// SIMATIC S7-200 project (STEP 7-Micro/WIN), CPU 226 REL 02.00

ORGANIZATION_BLOCK MAIN:OB1
TITLE=【PLC程序案例教程免烧砖机】
// 此PLC程序控制免烧砖机，包含生产控制和故障处理模块。 系统通过原料输送带、模具和成品输送带运行。
// 系统部署在生产车间，通过触摸屏操作界面进行参数设置和状态监控，支持手动和自动两种模式，满足不同操作需求。
// 
// 
// 操作员按下点动按钮可启动成品输送带。系统通过模式标志切换手动和自动模式：当模式标志为0时，系统处于手动模式；当模式标志为1时，系统处于自动模式。
// 在自动模式下，操作员按下启动按钮启动生产流程。系统首先检查生产批次计数器是否大于0，并确保到位传感器1、到位传感器3、到位传感器4和到位传感器5全部检测到位，只有这些条件满足时，状态变量才会从100变为58，进入生产状态。若任一传感器未就位，系统保持待机，避免设备运行风险。
// 生产开始后，原料通过输送带输入，随后进入布料阶段。布料过程被调用，当布料传感器检测到原料到位时，置位布料标志。在布料过程中，若布料标志置位，则激活布料执行信号。布料过程中，布料计数器记录布料次数。系统将布料计数器与布料上限计数器比较。若布料计数器小于布料上限计数器，布料继续；若达到上限，则根据布料模式变量切换布料逻辑，确保原料分配精准。
// 布料完成后，系统进入压制阶段，置位压制控制标志和压制执行信号。压制动作持续进行，直到到位传感器2检测到模具到位，随后压制执行信号复位。压制开始后，压制定时器1控制初始压制时间。随后，压制定时器2进一步控制压制时间，确保砖块成型质量稳定。压制结束后，成品通过成品输送带输出。压制计数器记录压制次数。系统将压制计数器与目标压制计数器比较以跟踪生产进度。
// 在手动模式下，操作员可通过点动按钮启动成品输送带。当到位传感器5置位时，成品输送带停止运行，以防止误操作导致设备损坏或安全事故。
// 系统还具备完善的故障监控功能。若故障总标志置位，表明某个环节出现异常，故障显示位1或故障显示位2会具体指示故障源，如执行机构1或2的异常状态。操作员可通过触摸屏查看详细故障信息并采取措施。
// 
BEGIN
Network 1 // 网络标题
// 网络注释
LD     SM0.1
CALL   SYSRESET:SBR13
Network 2
LDN    M31.0
CALL   Trouble_Display:SBR1
CALL   Run_Data_Change:SBR6
Network 3
LDN    M31.0
CALL   Trou_Run:SBR18
Network 4
LD     SM0.0
CALL   IOContral:SBR3
CALL   TOUCHER:SBR12
CALL   TOUCHER_Time:SBR10
CALL   TOUCHER_Time1:SBR11
CALL   SETUP_DATE:SBR19
Network 5
LDN    M3.2
AN     M31.0
CALL   Manual_batch:SBR4
CALL   Spot_Batch:SBR0
Network 6
LDN    M3.2
AN     M31.0
CALL   Manual_Spot:SBR17
Network 7
LD     M3.2
A      I2.3
AN     M31.0
CALL   AUTO_RESET:SBR5
CALL   Send_Take:SBR22
CALL   AUTO_PRODUCT:SBR15
Network 8
LDN    I4.0
CALL   Manual_batch1:SBR7
Network 9
LD     I4.0
CALL   AUTO1:SBR8
END_ORGANIZATION_BLOCK

SUBROUTINE_BLOCK Spot_Batch:SBR0
TITLE=子程序注释
BEGIN
Network 1 // 网络标题
// 网络注释
LDN    M4.4
AB=    VB742, 10
LD     I0.7
O      M22.5
ALD
AN     M8.0
S      M4.4, 1
S      M10.1, 1
Network 2
LD     M4.4
LDN    M22.5
AN     I0.7
O      M8.0
OB=    VB742, 0
ALD
R      M10.1, 1
R      M4.4, 1
Network 3
LDN    M4.7
AB=    VB742, 10
LD     I1.0
O      M22.6
ALD
AN     I3.2
S      M4.7, 1
S      M10.0, 1
Network 4
LD     M4.7
LDN    M22.6
AN     I1.0
O      I3.2
OB=    VB742, 0
ALD
R      M10.0, 1
R      M4.7, 1
Network 5
LDN    M5.1
LD     I0.5
O      M22.3
ALD
AB=    VB742, 10
AN     I2.4
AN     M8.2
S      M5.1, 1
S      M10.2, 1
Network 6
LD     M5.1
LDN    M22.3
AN     I0.5
O      M8.2
O      I2.4
OB=    VB742, 0
ALD
R      M10.2, 1
R      M5.1, 1
Network 7
LDN    M5.3
AB=    VB742, 10
LD     I0.6
O      M22.4
ALD
AN     I2.5
S      M5.3, 1
S      M10.4, 1
Network 8
LD     M5.3
LDN    M22.4
AN     I0.6
O      I2.5
OB=    VB742, 0
ALD
R      M10.4, 1
R      M5.3, 1
Network 9
LDN    M6.5
AB=    VB742, 10
LD     I1.1
O      M22.7
ALD
AN     I2.6
AN     M9.0
S      M6.5, 1
S      M11.4, 1
Network 10
LD     M6.5
LDN    M22.7
AN     I1.1
O      M9.0
O      I2.6
OB=    VB742, 0
ALD
R      M11.4, 1
R      M6.5, 1
Network 11
LDN    M6.7
AB=    VB742, 10
LD     I1.2
O      M23.0
ALD
AN     I2.7
AN     M9.1
S      M6.7, 1
S      M11.6, 1
Network 12
LD     M6.7
LDN    M23.0
AN     I1.2
O      M9.1
O      I2.7
OB=    VB742, 0
ALD
R      M11.6, 1
R      M6.7, 1
Network 13
LDN    M7.1
AB=    VB742, 10
LD     I1.3
O      M23.1
ALD
AN     I3.0
AN     M9.2
S      M7.1, 1
S      M12.1, 1
Network 14
LD     M7.1
LDN    M23.1
AN     I1.3
O      M9.2
O      I3.0
OB=    VB742, 0
ALD
R      M12.1, 1
R      M7.1, 1
Network 15
LDN    M7.3
AB=    VB742, 10
LD     I1.4
O      M23.2
ALD
AN     I3.1
AN     M9.3
S      M7.3, 1
S      M12.3, 1
Network 16
LD     M7.3
LDN    M23.2
AN     I1.4
O      M9.3
O      I3.1
OB=    VB742, 0
ALD
R      M12.3, 1
R      M7.3, 1
Network 17
LDN    M7.5
AB=    VB742, 10
LD     I1.5
O      M23.3
ALD
AN     I2.7
AN     M12.6
S      M7.5, 1
S      M12.0, 1
Network 18
LD     M7.5
LDN    M23.3
AN     I1.5
O      M12.6
O      I2.7
OB=    VB742, 0
ALD
R      M12.0, 1
R      M7.5, 1
END_SUBROUTINE_BLOCK

SUBROUTINE_BLOCK Trouble_Display:SBR1
TITLE=
BEGIN
Network 1
LD     I0.7
O      M22.5
AN     I2.5
AN     V5000.3
AB=    VB742, 0
=      V5000.3
Network 2
LD     I1.0
O      M22.6
A      I3.2
AN     V5000.4
=      V5000.4
Network 3
LD     I0.5
O      M22.3
LD     I2.4
ON     I3.2
ON     I2.6
ON     I3.1
ALD
AN     V5000.5
AB=    VB742, 0
=      V5000.5
Network 4
LD     I0.6
O      M22.4
LDN    I2.6
O      I2.5
ALD
AN     V5000.6
AB=    VB742, 0
=      V5000.6
Network 5
LD     I1.1
O      M22.7
A      I2.6
AN     V5001.3
=      V5001.3
Network 6
LD     I1.2
O      M23.0
LDN    I2.5
O      I2.7
ALD
AN     V5001.4
AB=    VB742, 0
=      V5001.4
Network 7
LD     I1.5
O      M23.3
LDN    I2.5
O      I2.7
ALD
AN     V5001.5
AB=    VB742, 0
=      V5001.5
Network 8
LD     I1.4
O      M23.2
A      I3.1
AN     V5001.6
=      V5001.6
Network 9
LD     I1.3
O      M23.1
LDN    I2.5
O      I3.0
ALD
AN     V5001.7
AB=    VB742, 0
=      V5001.7
Network 10
LD     I0.5
O      M22.3
LD     I0.6
O      M22.4
ALD
=      V5003.3
Network 11
LD     I1.1
O      M22.7
LD     I1.2
O      M23.0
ALD
=      V5003.4
Network 12
LD     I1.3
O      M23.1
LD     I1.4
O      M23.2
ALD
=      V5003.5
END_SUBROUTINE_BLOCK

SUBROUTINE_BLOCK RESET:SBR2
TITLE=
BEGIN
Network 1
LD     SM0.0
R      M3.3, 1
Network 2
LD     SM0.0
MOVB   100, VB700
MOVB   100, VB702
Network 3
LD     SM0.0
MOVB   0, QB0
MOVB   0, QB2
Network 4
LD     SM0.0
R      Q1.3, 1
R      Q1.4, 1
R      Q1.5, 1
R      Q1.6, 1
R      Q1.7, 1
Network 5
LD     SM0.0
MOVW   +0, VW802
MOVW   +0, VW806
MOVW   +0, VW812
Network 6
LD     SM0.0
R      M10.0, 6
R      M11.4, 4
R      M12.0, 8
R      M30.0, 1
R      M18.1, 1
R      M18.4, 1
R      M28.7, 1
Network 7
LD     SM0.0
R      M18.7, 1
R      V5003.7, 3
R      M21.0, 4
R      V5003.1, 2
R      M2.3, 1
Network 8
LD     SM0.0
R      M2.0, 3
R      M4.4, 1
R      M4.7, 1
R      M5.1, 1
R      M5.3, 1
R      M6.5, 1
R      M6.7, 1
R      M7.1, 1
R      M7.3, 1
R      M7.5, 1
R      M18.0, 2
R      M18.5, 1
Network 9
LD     SM0.0
R      M4.2, 1
R      M4.5, 1
R      M5.0, 1
R      M5.2, 1
R      M6.4, 1
R      M6.6, 1
R      M7.0, 1
R      M7.2, 1
R      M7.6, 1
R      M12.7, 1
R      M7.4, 1
R      M7.7, 1
R      M18.2, 3
R      M4.3, 1
R      M4.6, 1
Network 10
LD     SM0.0
R      M21.6, 1
R      M29.0, 8
R      M30.3, 5
END_SUBROUTINE_BLOCK

SUBROUTINE_BLOCK IOContral:SBR3
TITLE=
BEGIN
Network 1
LD     SM0.0
TODR   VB5100
BMB    VB5100, VB2450, 8
Network 2
LD     SM0.0
LPS
A      M31.1
AW<=   VW94, VW82
R      M31.0, 1
LRD
A      M31.1
AW>    VW94, VW82
S      M31.0, 1
LRD
A      M31.2
AW<=   VW94, VW86
R      M31.0, 1
LRD
A      M31.2
AW>    VW94, VW86
S      M31.0, 1
LPP
AW=    VW90, +370
R      M31.0, 1
Network 3
LDW>=  VW804, +1
MOVW   VW804, VW800
-I     +1, VW800
Network 4
LDB=   QB0, 0
MOVW   +0, VW144
MOVW   +0, VW146
Network 5
LD     I2.3
A      Q1.2
MOVW   VW144, VW136
*I     VW152, VW136
MOVW   VW146, VW138
*I     VW148, VW138
Network 6
LD     M4.0
LD     I0.4
O      M22.2
ALD
ED
R      M4.0, 2
R      Q1.2, 1
Network 7
LD     M4.0
A      M4.1
AN     I2.3
R      M4.0, 2
R      Q1.2, 1
S      M3.0, 1
R      M3.1, 1
CALL   RESET:SBR2
Network 8
LD     Q1.2
A      I2.3
AN     M4.1
S      M4.1, 1
Network 9
LDN    M4.0
AN     I2.3
LD     I0.4
O      M22.2
ALD
ED
S      M4.0, 1
S      Q1.2, 1
Network 10
LD     I2.3
A      Q1.2
MOVW   VW136, AQW0
MOVW   VW138, AQW2
Network 11
LD     M31.0
LD     I0.3
O      I0.5
O      I0.6
O      I0.7
O      I1.0
O      I1.1
O      I1.2
O      I1.3
O      I1.4
O      I1.5
O      I1.6
O      I1.7
O      I2.0
O      I2.1
ALD
=      V5005.4
Network 12
LDN    M31.0
A      I0.0
AN     I2.3
LD     I0.3
O      I0.5
O      I0.6
O      I0.7
O      I1.0
O      I1.1
O      I1.2
O      I1.3
O      I1.4
O      I1.5
ALD
=      V5005.3
Network 13
LDN    M31.0
AN     M3.1
AN     V5003.6
LD     I0.3
O      M22.1
ALD
LD     M3.3
ON     M3.2
ON     I2.5
ON     I2.3
ON     I3.3
ON     I2.6
ON     I3.1
ALD
=      V5003.6
Network 14
LDW<>  VW90, +370
AN     M28.5
A      M28.6
LPS
INCW   VW1006
AENO
MOVW   VW1006, VW94
LRD
S      M28.5, 1
LPP
R      M28.6, 1
Network 15
LD     M28.5
AN     SM31.7
R      SM31.0, 1
S      SM31.1, 1
MOVW   +94, SMW32
S      SM31.7, 1
R      M28.5, 1
Network 16
LD     M3.6
R      M3.1, 1
S      M3.0, 1
R      M3.6, 1
CALL   RESET:SBR2
Network 17
LD     M3.5
R      M3.5, 1
CALL   RESET:SBR2
Network 18
LD     M3.1
LD     M9.3
O      M8.1
O      M8.2
O      M8.3
O      M9.0
O      M9.2
O      M12.6
O      M9.7
O      M9.1
ALD
S      M3.0, 1
R      M3.1, 1
CALL   RESET:SBR2
Network 19
LD     M3.7
AN     I4.0
CALL   RESET1:SBR9
Network 20
LDN    I0.0
S      M3.4, 1
Network 21
LD     I0.0
LPS
R      M3.4, 1
EU
S      M3.5, 1
LPP
ED
S      M3.6, 1
Network 22
LDN    M3.4
S      M3.2, 1
Network 23
LD     M3.4
R      M3.2, 1
Network 24
LDN    I4.0
R      M3.7, 1
Network 25
LD     I4.0
S      M3.7, 1
END_SUBROUTINE_BLOCK

SUBROUTINE_BLOCK Manual_batch:SBR4
TITLE=
BEGIN
Network 1
LD     I0.2
O      M22.0
CALL   RESET:SBR2
Network 2
LD     M4.2
AB=    VB742, 0
A      Q0.3
LD     I0.7
O      M22.5
ALD
ED
R      M10.1, 1
R      M4.2, 1
Network 3
LD     M4.2
A      Q0.3
LD     M8.0
ON     I2.5
O      I1.0
OB=    VB742, 10
O      M22.6
ALD
R      M10.1, 1
R      M4.2, 1
Network 4
LDN    M4.2
AN     M4.3
A      I2.5
AB=    VB742, 0
AN     M8.0
AN     M22.6
AN     I1.0
LD     I0.7
O      M22.5
ALD
ED
S      M4.2, 1
S      M10.1, 1
R      T163, 1
Network 5
LD     M4.5
AB=    VB742, 0
A      Q0.2
LD     I1.0
O      M22.6
ALD
ED
R      M10.0, 1
R      M4.5, 1
Network 6
LD     M4.5
A      Q0.2
LD     I3.2
O      M8.1
O      I0.7
OB=    VB742, 10
O      M22.5
ALD
R      M10.0, 1
R      M4.5, 1
Network 7
LDN    M4.5
AN     M4.3
AN     M22.5
AN     I0.7
AB=    VB742, 0
AN     M8.1
AN     I3.2
LD     I1.0
O      M22.6
ALD
ED
S      M4.5, 1
S      M10.0, 1
Network 8
LD     M5.0
AB=    VB742, 0
A      Q0.1
LD     I0.5
O      M22.3
ALD
ED
R      M10.2, 1
R      M5.0, 1
Network 9
LD     M5.0
A      Q0.1
LD     I2.4
O      M8.2
O      M22.4
ON     I3.2
ON     I2.6
ON     I3.1
O      I0.6
OB=    VB742, 10
ALD
R      M10.2, 1
R      M5.0, 1
Network 10
LDN    M5.0
AB=    VB742, 0
A      I3.2
A      I2.6
A      I3.1
AN     M22.4
AN     I0.6
AN     I2.4
AN     M8.2
LD     I0.5
O      M22.3
ALD
ED
S      M5.0, 1
S      M10.2, 1
Network 11
LD     M5.2
AB=    VB742, 0
A      Q0.0
LD     I0.6
O      M22.4
ALD
ED
R      M10.4, 1
R      M5.2, 1
Network 12
LD     M5.2
A      Q0.0
LD     I2.5
O      M8.3
ON     I2.6
O      I0.5
OB=    VB742, 10
O      M22.3
ALD
R      M10.4, 1
R      M5.2, 1
Network 13
LDN    M5.2
AB=    VB742, 0
A      I2.6
AN     I2.5
AN     M22.3
AN     I0.5
AN     M8.3
LD     I0.6
O      M22.4
ALD
ED
S      M5.2, 1
S      M10.4, 1
Network 14
LD     M6.4
AB=    VB742, 0
A      Q0.4
LD     I1.1
O      M22.7
ALD
ED
R      M11.4, 1
R      M6.4, 1
Network 15
LD     M6.4
A      Q0.4
LD     I2.6
O      M9.0
O      I1.2
OB=    VB742, 10
O      M23.0
ALD
R      M11.4, 1
R      M6.4, 1
Network 16
LDN    M6.4
AB=    VB742, 0
AN     I2.6
AN     M23.0
AN     I1.2
AN     M9.0
LD     I1.1
O      M22.7
ALD
ED
S      M6.4, 1
S      M11.4, 1
Network 17
LD     M6.6
AB=    VB742, 0
A      Q0.5
LD     I1.2
O      M23.0
ALD
ED
R      M11.6, 1
R      M6.6, 1
Network 18
LD     M6.6
A      Q0.5
LD     I2.7
OB=    VB742, 10
O      M9.1
ON     I2.5
O      M22.7
O      I1.1
ALD
R      M11.6, 1
R      M6.6, 1
Network 19
LDN    M6.6
AB=    VB742, 0
A      I2.5
AN     I2.7
AN     M22.7
AN     I1.1
AN     M9.1
LD     I1.2
O      M23.0
ALD
ED
S      M6.6, 1
S      M11.6, 1
Network 20
LD     M7.0
AB=    VB742, 0
A      Q0.6
LD     I1.3
O      M23.1
ALD
ED
R      M12.1, 1
R      M7.0, 1
Network 21
LD     M7.0
A      Q0.6
LD     I1.4
O      M9.2
ON     I2.5
O      M23.2
O      I3.0
OB=    VB742, 10
ALD
R      M12.1, 1
R      M7.0, 1
Network 22
LDN    M7.0
AB=    VB742, 0
AN     M23.2
AN     I1.4
A      I2.5
AN     I3.0
AN     M9.2
LD     I1.3
O      M23.1
ALD
ED
S      M7.0, 1
S      M12.1, 1
Network 23
LD     M7.2
AB=    VB742, 0
A      Q0.7
LD     I1.4
O      M23.2
ALD
ED
R      M12.3, 1
R      M7.2, 1
Network 24
LD     M7.2
A      Q0.7
LD     I1.3
O      M9.3
O      I3.1
OB=    VB742, 10
O      M23.1
ALD
R      M12.3, 1
R      M7.2, 1
Network 25
LDN    M7.2
AB=    VB742, 0
AN     M23.1
AN     I1.3
AN     I3.1
AN     M9.3
LD     I1.4
O      M23.2
ALD
ED
S      M7.2, 1
S      M12.3, 1
Network 26
LD     M7.4
AB=    VB742, 0
A      Q0.5
LD     I1.5
O      M23.3
ALD
ED
R      M12.0, 1
R      M7.4, 1
Network 27
LD     M7.4
A      Q0.5
LD     M12.6
O      I1.1
ON     I2.5
O      M22.7
O      I2.7
OB=    VB742, 10
ALD
R      M12.0, 1
R      M7.4, 1
Network 28
LDN    M7.4
AN     M22.7
AN     I1.1
AB=    VB742, 0
A      I2.5
AN     M12.6
AN     I2.7
LD     I1.5
O      M23.3
ALD
ED
S      M7.4, 1
S      M12.0, 1
END_SUBROUTINE_BLOCK

SUBROUTINE_BLOCK AUTO_RESET:SBR5
TITLE=
BEGIN
Network 1
LD     I0.2
LDN    I2.5
ON     I3.3
ON     I3.2
ON     I2.6
ON     I3.1
O      M3.1
ALD
CALL   RESET:SBR2
MOVB   90, VB700
S      M3.0, 1
R      M3.1, 1
Network 2
LDB=   VB700, 90
TON    T160, +5
A      T160
R      T160, 1
MOVB   100, VB700
Network 3
LDB=   VB700, 90
LDN    I2.5
ON     I3.2
ON     I2.6
ON     I3.1
ON     I3.3
ALD
MOVB   85, VB700
Network 4
LDB=   VB700, 85
S      M11.4, 1
A      I2.6
R      M11.4, 1
MOVB   80, VB700
Network 5
LDB=   VB700, 80
S      M10.0, 1
A      I3.2
R      M10.0, 1
MOVB   75, VB700
Network 6
LDB=   VB700, 75
S      M10.4, 1
A      I2.5
R      M10.4, 1
MOVB   72, VB700
Network 7
LDB=   VB700, 72
S      Q1.5, 1
A      I3.3
R      Q1.5, 1
MOVB   66, VB700
Network 8
LDB=   VB700, 66
S      M12.3, 1
A      I3.1
R      M12.3, 1
MOVB   90, VB700
Network 9
LDB=   VB700, 66
CRET
END_SUBROUTINE_BLOCK

SUBROUTINE_BLOCK Run_Data_Change:SBR6
TITLE=
BEGIN
Network 1
LD     M10.0
A      M19.0
A      M19.1
AN     M8.1
MOVW   VW396, VW144
MOVW   VW400, VW146
TON    T136, VW212
A      T136
R      T136, 1
S      M8.1, 1
S      V5002.4, 1
Network 2
LD     M10.0
A      M19.0
AN     M19.1
MOVW   VW394, VW144
MOVW   VW398, VW146
TON    T43, VW210
A      T43
R      T43, 1
S      M19.1, 1
Network 3
LD     M10.0
S      Q0.2, 1
AN     M19.0
AN     M19.1
MOVW   VW392, VW144
MOVW   VW398, VW146
TON    T42, VW208
A      T42
R      T42, 1
S      M19.0, 1
Network 4
LDN    M10.0
R      Q0.2, 1
R      M19.0, 2
R      M8.1, 1
Network 5
LD     M10.1
A      M19.2
A      M19.3
AN     M8.0
MOVW   VW384, VW144
MOVW   VW388, VW146
TON    T134, VW204
A      T134
R      T134, 1
S      M8.0, 1
S      V5002.3, 1
Network 6
LD     M10.1
A      M19.2
AN     M19.3
MOVW   VW382, VW144
MOVW   VW386, VW146
TON    T41, VW202
A      T41
R      T41, 1
S      M19.3, 1
Network 7
LD     M10.1
S      Q0.3, 1
AN     M19.2
AN     M19.3
MOVW   VW380, VW144
MOVW   VW386, VW146
TON    T40, VW200
A      T40
R      T40, 1
S      M19.2, 1
Network 8
LDN    M10.1
R      Q0.3, 1
R      M19.2, 2
R      M8.0, 1
Network 9
LD     M10.2
A      M10.3
A      M19.4
AN     M8.2
MOVW   VW408, VW144
MOVW   VW412, VW146
TON    T130, VW220
A      T130
R      T130, 1
S      M8.2, 1
S      V5002.1, 1
Network 10
LD     M10.2
A      M10.3
AN     M19.4
MOVW   VW406, VW144
MOVW   VW410, VW146
TON    T45, VW218
A      T45
R      T45, 1
S      M19.4, 1
Network 11
LD     M10.2
O      M18.1
S      Q0.1, 1
Network 12
LD     M10.2
AN     M10.3
AN     M19.4
MOVW   VW404, VW144
MOVW   VW410, VW146
TON    T44, VW216
A      T44
R      T44, 1
S      M10.3, 1
Network 13
LDN    M10.2
LPS
AN     M18.1
R      Q0.1, 1
LRD
R      M10.3, 1
LRD
R      M19.4, 1
LPP
R      M8.2, 1
Network 14
LD     M10.4
A      M10.5
A      M19.5
AN     M8.3
MOVW   VW420, VW144
MOVW   VW424, VW146
TON    T132, VW228
A      T132
R      T132, 1
S      M8.3, 1
S      V5002.2, 1
Network 15
LD     M10.4
A      M10.5
AN     M19.5
MOVW   VW418, VW144
MOVW   VW422, VW146
TON    T47, VW226
A      T47
R      T47, 1
S      M19.5, 1
Network 16
LD     M10.4
O      M18.4
S      Q0.0, 1
Network 17
LD     M10.4
AN     M10.5
AN     M19.5
MOVW   VW416, VW144
MOVW   VW422, VW146
TON    T46, VW224
A      T46
R      T46, 1
S      M10.5, 1
Network 18
LDN    M10.4
LPS
AN     M18.4
R      Q0.0, 1
LRD
R      M10.5, 1
LRD
R      M19.5, 1
LPP
R      M8.3, 1
Network 19
LD     M11.4
A      M11.5
A      M20.4
AN     M9.0
MOVW   VW480, VW144
MOVW   VW484, VW146
TON    T138, VW268
A      T138
R      T138, 1
S      M9.0, 1
S      V5002.5, 1
Network 20
LD     M11.4
A      M11.5
AN     M20.4
MOVW   VW478, VW144
MOVW   VW482, VW146
TON    T57, VW266
A      T57
R      T57, 1
S      M20.4, 1
Network 21
LD     M11.4
S      Q0.4, 1
AN     M11.5
AN     M20.4
MOVW   VW476, VW144
MOVW   VW482, VW146
TON    T56, VW264
A      T56
R      T56, 1
S      M11.5, 1
Network 22
LDN    M11.4
R      Q0.4, 1
R      M11.5, 1
R      M20.4, 1
R      M9.0, 1
Network 23
LD     M11.6
A      M11.7
A      M20.5
AN     M9.1
MOVW   VW492, VW144
MOVW   VW496, VW146
TON    T140, VW276
A      T140
R      T140, 1
S      M9.1, 1
Network 24
LD     M11.6
O      M12.0
S      Q0.5, 1
Network 25
LD     M11.6
A      M11.7
AN     M20.5
MOVW   VW490, VW144
MOVW   VW494, VW146
TON    T59, VW274
A      T59
R      T59, 1
S      M20.5, 1
Network 26
LD     M11.6
AN     M11.7
AN     M20.5
MOVW   VW488, VW144
MOVW   VW494, VW146
TON    T58, VW272
A      T58
R      T58, 1
S      M11.7, 1
Network 27
LDN    M11.6
LPS
AN     M12.0
R      Q0.5, 1
LRD
R      M11.7, 1
LRD
R      M20.5, 1
LPP
R      M9.1, 1
Network 28
LD     M12.1
A      M12.2
A      M20.6
AN     M9.2
MOVW   VW504, VW144
MOVW   VW508, VW146
TON    T142, VW284
A      T142
R      T142, 1
S      M9.2, 1
S      V5002.7, 1
Network 29
LD     M12.1
A      M12.2
AN     M20.6
MOVW   VW502, VW144
MOVW   VW506, VW146
TON    T61, VW282
A      T61
R      T61, 1
S      M20.6, 1
Network 30
LD     M12.1
O      M30.0
S      Q0.6, 1
Network 31
LD     M12.1
AN     M12.2
AN     M20.6
MOVW   VW500, VW144
MOVW   VW506, VW146
TON    T60, VW280
A      T60
R      T60, 1
S      M12.2, 1
Network 32
LDN    M12.1
LPS
AN     M30.0
R      Q0.6, 1
LRD
R      M12.2, 1
LRD
R      M20.6, 1
LPP
R      M9.2, 1
Network 33
LD     M12.3
A      M12.4
A      M20.7
AN     M9.3
MOVW   VW516, VW144
MOVW   VW520, VW146
TON    T144, VW292
A      T144
R      T144, 1
S      M9.3, 1
S      V5003.0, 1
Network 34
LD     M12.3
A      M12.4
AN     M20.7
MOVW   VW514, VW144
MOVW   VW518, VW146
TON    T63, VW290
A      T63
R      T63, 1
S      M20.7, 1
Network 35
LD     M12.3
S      Q0.7, 1
AN     M12.4
AN     M20.7
MOVW   VW512, VW144
MOVW   VW518, VW146
TON    T62, VW288
A      T62
R      T62, 1
S      M12.4, 1
Network 36
LDN    M12.3
R      Q0.7, 1
R      M12.4, 1
R      M20.7, 1
R      M9.3, 1
Network 37
LD     M12.0
MOVW   VW524, VW144
MOVW   VW526, VW146
Network 38
LD     M18.1
O      M18.4
MOVW   VW540, VW144
MOVW   VW542, VW146
Network 39
LD     M30.0
A      M30.1
A      M30.2
AN     M9.7
MOVW   VW534, VW144
MOVW   VW538, VW146
TON    T167, VW284
A      T167
R      T167, 1
S      M9.7, 1
S      V5002.7, 1
Network 40
LD     M30.0
A      M30.1
AN     M30.2
MOVW   VW532, VW144
MOVW   VW536, VW146
TON    T166, VW282
A      T166
R      T166, 1
S      M30.2, 1
Network 41
LD     M30.0
AN     M30.1
AN     M30.2
MOVW   VW530, VW144
MOVW   VW536, VW146
TON    T165, VW280
A      T165
R      T165, 1
S      M30.1, 1
Network 42
LDN    M30.0
R      M30.1, 2
R      M9.7, 1
END_SUBROUTINE_BLOCK

SUBROUTINE_BLOCK Manual_batch1:SBR7
TITLE=
BEGIN
Network 1
LD     M1.0
A      Q2.0
LD     I5.2
O      M24.6
ALD
ED
R      Q2.0, 1
R      M1.0, 1
Network 2
LD     M1.0
A      Q2.0
LD     I4.2
O      M24.7
O      I5.3
ALD
R      Q2.0, 1
R      M1.0, 1
Network 3
LDN    M1.0
AN     I4.2
AN     M24.7
AN     I5.3
LD     I5.2
O      M24.6
ALD
ED
S      M1.0, 1
S      Q2.0, 1
Network 4
LD     M1.2
A      Q2.1
LD     I5.3
O      M24.7
ALD
ED
R      Q2.1, 1
R      M1.2, 1
R      Q2.2, 1
R      M25.5, 1
R      M25.4, 1
Network 5
LD     M1.2
A      Q2.1
LD     M25.7
O      M25.5
ALD
S      Q2.2, 1
Network 6
LD     M1.2
A      Q2.1
LD     I4.3
O      M24.6
O      I5.2
ALD
R      Q2.1, 1
R      M1.2, 1
R      Q2.2, 1
R      M25.7, 1
R      M25.5, 1
R      M25.4, 1
Network 7
LDN    M1.2
AN     I4.3
AN     M24.6
AN     I5.2
LD     I5.3
O      M24.7
ALD
ED
S      M1.2, 1
S      Q2.1, 1
Network 8
LD     M1.4
A      Q1.0
LD     I5.0
O      M24.4
ALD
ED
R      Q1.0, 1
R      M1.4, 1
R      M9.4, 1
Network 9
LD     M1.4
A      Q1.0
LD     I4.5
O      M24.5
O      I5.1
O      M9.4
ALD
R      Q1.0, 1
R      M1.4, 1
R      M9.4, 1
Network 10
LDN    M1.4
AN     I4.5
AN     M9.4
AN     M24.5
AN     I5.1
LD     I5.0
O      M24.4
ALD
ED
S      M1.4, 1
S      Q1.0, 1
Network 11
LD     M1.6
A      Q1.1
LD     I5.1
O      M24.5
ALD
ED
R      Q1.1, 1
R      M1.6, 1
Network 12
LD     M1.6
A      Q1.1
LD     I4.6
O      M24.4
O      I5.0
ALD
R      Q1.1, 1
R      M1.6, 1
Network 13
LDN    M1.6
AN     I4.6
AN     M24.4
AN     I5.0
LD     I5.1
O      M24.5
ALD
ED
S      M1.6, 1
S      Q1.1, 1
Network 14
LDN    M25.4
AN     M25.5
AN     M25.7
A      Q2.1
TON    T154, VW62
A      T154
R      T154, 1
S      M25.7, 1
S      M25.4, 1
Network 15
LD     M25.7
TON    T155, VW54
A      T155
R      T155, 1
R      M25.7, 1
R      Q2.2, 1
Network 16
LD     SM0.0
LPS
AN     I4.7
MOVW   +0, VW828
LPP
AW>=   VW66, +1
AN     Q2.1
MOVW   VW828, VW64
*I     VW60, VW64
AW<=   VW64, VW58
MOVW   VW58, VW62
-I     VW64, VW62
Network 17
LD     SM0.0
LPS
A      Q2.1
S      M25.6, 1
LPP
A      I4.7
A      M25.6
A      I4.3
EU
R      M25.6, 1
INCW   VW828
Network 18
LD     I4.4
A      Q2.1
S      M25.5, 1
R      T154, 1
R      M25.7, 1
R      T155, 1
Network 19
LD     SM0.0
MOVW   VW824, VW66
-I     VW828, VW66
END_SUBROUTINE_BLOCK

SUBROUTINE_BLOCK AUTO1:SBR8
TITLE=
BEGIN
Network 1
LDB=   VB701, 100
AW<    VW828, VW824
AN     M3.3
A      I4.1
A      I4.6
MOVB   90, VB701
Network 2
LDB=   VB701, 90
S      Q2.0, 1
R      T157, 1
MOVB   88, VB701
Network 3
LDB=   VB701, 88
TON    T157, VW74
A      T157
R      T157, 1
S      Q2.2, 1
MOVB   86, VB701
Network 4
LDB=   VB701, 88
A      I4.2
R      T157, 1
R      Q2.2, 1
MOVB   86, VB701
Network 5
LDB=   VB701, 86
OB=    VB701, 88
AN     I4.1
R      Q2.2, 1
Network 6
LDB=   VB701, 86
A      I4.2
MOVB   85, VB701
Network 7
LDB=   VB701, 85
TON    T210, +1
A      T210
LPS
R      T210, 1
AN     I4.2
MOVB   86, VB701
LPP
A      I4.2
R      Q2.0, 1
MOVB   83, VB701
Network 8
LDB=   VB701, 83
TON    T218, +5
A      T218
R      T218, 1
MOVB   80, VB701
Network 9
LDB=   VB701, 80
S      Q1.0, 1
A      I4.5
MOVB   75, VB701
Network 10
LDB=   VB701, 75
TON    T211, +1
A      T211
LPS
R      T211, 1
AN     I4.5
MOVB   80, VB701
LPP
A      I4.5
R      Q1.0, 1
R      M9.4, 1
MOVB   73, VB701
Network 11
LDB=   VB701, 75
A      M9.4
R      Q1.0, 1
R      M9.4, 1
MOVB   73, VB701
Network 12
LDB=   VB701, 73
A      I4.5
MOVB   72, VB701
Network 13
LDB=   VB701, 72
TON    T212, +5
A      T212
R      T212, 1
MOVB   70, VB701
Network 14
LDB=   VB701, 70
S      Q2.1, 1
AN     M21.4
A      Q2.1
TON    T153, VW62
A      T153
R      T153, 1
S      Q2.2, 1
S      M21.4, 1
S      M21.3, 1
Network 15
LDB=   VB701, 70
LPS
A      I4.4
MOVB   69, VB701
LPP
A      I4.3
MOVB   67, VB701
Network 16
LDB=   VB701, 69
TON    T213, +1
A      T213
R      T213, 1
S      Q2.2, 1
R      T126, 1
R      T153, 1
S      Q2.1, 1
MOVB   68, VB701
Network 17
LDB=   VB701, 68
A      I4.3
MOVB   67, VB701
Network 18
LDB=   VB701, 67
TON    T214, +1
A      T214
LPS
R      T214, 1
A      I4.3
MOVB   65, VB701
LPP
AN     I4.3
MOVB   70, VB701
S      Q2.1, 1
S      Q2.2, 1
Network 19
LDB=   VB701, 65
R      Q2.1, 1
R      M21.3, 1
R      Q2.2, 1
R      M21.4, 1
Network 20
LDB=   VB701, 65
LPS
AN     I4.7
MOVB   64, VB701
LPP
A      I4.7
INCW   VW828
AW>=   VW828, VW824
S      M3.3, 1
S      V5005.2, 1
S      M31.6, 1
R      T161, 1
Network 21
LDB=   VB701, 65
A      I4.7
MOVB   64, VB701
Network 22
LDB=   VB701, 64
TON    T215, +5
A      T215
R      T215, 1
MOVB   60, VB701
Network 23
LDB=   VB701, 60
S      Q1.1, 1
A      I4.6
MOVB   55, VB701
Network 24
LDB=   VB701, 55
TON    T216, +1
A      T216
LPS
R      T216, 1
A      I4.6
R      Q1.1, 1
MOVB   50, VB701
LPP
AN     I4.6
MOVB   60, VB701
Network 25
LDB=   VB701, 50
A      I4.6
MOVB   45, VB701
Network 26
LDB=   VB701, 45
TON    T217, +5
A      T217
R      T217, 1
MOVB   100, VB701
Network 27
LD     M21.3
TON    T126, VW54
A      T126
R      T126, 1
R      M21.3, 1
R      Q2.2, 1
Network 28
LDN    I4.7
A      M31.6
TON    T161, +10
A      T161
R      T161, 1
R      M3.3, 1
R      V5005.2, 1
R      M31.6, 1
MOVW   +0, VW828
Network 29
LD     SM0.0
MOVW   VW824, VW66
-I     VW828, VW66
Network 30
LD     SM0.0
AW>=   VW66, +1
AN     Q2.1
MOVW   VW828, VW64
*I     VW60, VW64
AW<=   VW64, VW58
MOVW   VW58, VW62
-I     VW64, VW62
Network 31
LD     SM0.0
AN     I4.7
R      M3.3, 1
MOVW   +0, VW828
END_SUBROUTINE_BLOCK

SUBROUTINE_BLOCK RESET1:SBR9
TITLE=
BEGIN
Network 1
LD     SM0.0
R      M1.0, 8
R      M21.4, 1
R      Q1.0, 2
R      Q2.0, 3
R      M9.4, 1
R      V5005.7, 1
R      M25.7, 1
R      M25.6, 1
R      M25.5, 1
R      M21.3, 1
R      M25.4, 1
Network 2
LD     SM0.0
MOVB   100, VB701
END_SUBROUTINE_BLOCK

SUBROUTINE_BLOCK TOUCHER_Time:SBR10
TITLE=
BEGIN
Network 1
LDW<>  VW2360, VW540
MOVW   VW2360, VW540
Network 2
LDW<>  VW2362, VW542
MOVW   VW2362, VW542
Network 3
LD     SM0.0
MOVR   VD3070, VD3500
*R     10.0, VD3500
ROUND  VD3500, VD3500
Network 4
LDD<>  VD3500, VD2070
MOVD   VD3500, VD2070
DTI    VD3500, VW200
Network 5
LD     SM0.0
MOVR   VD3074, VD3504
*R     10.0, VD3504
ROUND  VD3504, VD3504
Network 6
LDD<>  VD3504, VD2074
MOVD   VD3504, VD2074
DTI    VD3504, VW202
Network 7
LD     SM0.0
MOVR   VD3078, VD3508
*R     10.0, VD3508
ROUND  VD3508, VD3508
Network 8
LDD<>  VD3508, VD2078
MOVD   VD3508, VD2078
DTI    VD3508, VW204
Network 9
LD     SM0.0
MOVR   VD3086, VD3512
*R     10.0, VD3512
ROUND  VD3512, VD3512
Network 10
LDD<>  VD3512, VD2086
MOVD   VD3512, VD2086
DTI    VD3512, VW208
Network 11
LD     SM0.0
MOVR   VD3090, VD3516
*R     10.0, VD3516
ROUND  VD3516, VD3516
Network 12
LDD<>  VD3516, VD2090
MOVD   VD3516, VD2090
DTI    VD3516, VW210
Network 13
LD     SM0.0
MOVR   VD3094, VD3520
*R     10.0, VD3520
ROUND  VD3520, VD3520
Network 14
LDD<>  VD3520, VD2094
MOVD   VD3520, VD2094
DTI    VD3520, VW212
Network 15
LD     SM0.0
MOVR   VD3102, VD3524
*R     10.0, VD3524
ROUND  VD3524, VD3524
Network 16
LDD<>  VD3524, VD2102
MOVD   VD3524, VD2102
DTI    VD3524, VW216
Network 17
LD     SM0.0
MOVR   VD3106, VD3528
*R     10.0, VD3528
ROUND  VD3528, VD3528
Network 18
LDD<>  VD3528, VD2106
MOVD   VD3528, VD2106
DTI    VD3528, VW218
Network 19
LD     SM0.0
MOVR   VD3110, VD3532
*R     10.0, VD3532
ROUND  VD3532, VD3532
Network 20
LDD<>  VD3532, VD2110
MOVD   VD3532, VD2110
DTI    VD3532, VW220
Network 21
LD     SM0.0
MOVR   VD3118, VD3536
*R     10.0, VD3536
ROUND  VD3536, VD3536
Network 22
LDD<>  VD3536, VD2118
MOVD   VD3536, VD2118
DTI    VD3536, VW224
Network 23
LD     SM0.0
MOVR   VD3122, VD3540
*R     10.0, VD3540
ROUND  VD3540, VD3540
Network 24
LDD<>  VD3540, VD2122
MOVD   VD3540, VD2122
DTI    VD3540, VW226
Network 25
LD     SM0.0
MOVR   VD3126, VD3544
*R     10.0, VD3544
ROUND  VD3544, VD3544
Network 26
LDD<>  VD3544, VD2126
MOVD   VD3544, VD2126
DTI    VD3544, VW228
Network 27
LD     SM0.0
MOVR   VD3196, VD3596
*R     10.0, VD3596
ROUND  VD3596, VD3596
Network 28
LDD<>  VD3596, VD1196
MOVD   VD3596, VD1196
DTI    VD3596, VW264
Network 29
LD     SM0.0
MOVR   VD3200, VD3600
*R     10.0, VD3600
ROUND  VD3600, VD3600
Network 30
LDD<>  VD3600, VD1200
MOVD   VD3600, VD1200
DTI    VD3600, VW266
Network 31
LD     SM0.0
MOVR   VD3204, VD3604
*R     10.0, VD3604
ROUND  VD3604, VD3604
Network 32
LDD<>  VD3604, VD1204
MOVD   VD3604, VD1204
DTI    VD3604, VW268
END_SUBROUTINE_BLOCK

SUBROUTINE_BLOCK TOUCHER_Time1:SBR11
TITLE=
BEGIN
Network 1
LD     SM0.0
MOVR   VD3212, VD3608
*R     10.0, VD3608
ROUND  VD3608, VD3608
Network 2
LDD<>  VD3608, VD1212
MOVD   VD3608, VD1212
DTI    VD3608, VW272
Network 3
LD     SM0.0
MOVR   VD3216, VD3612
*R     10.0, VD3612
ROUND  VD3612, VD3612
Network 4
LDD<>  VD3612, VD1216
MOVD   VD3612, VD1216
DTI    VD3612, VW274
Network 5
LD     SM0.0
MOVR   VD3220, VD3616
*R     10.0, VD3616
ROUND  VD3616, VD3616
Network 6
LDD<>  VD3616, VD1220
MOVD   VD3616, VD1220
DTI    VD3616, VW276
Network 7
LD     SM0.0
MOVR   VD3228, VD3620
*R     10.0, VD3620
ROUND  VD3620, VD3620
Network 8
LDD<>  VD3620, VD1228
MOVD   VD3620, VD1228
DTI    VD3620, VW280
Network 9
LD     SM0.0
MOVR   VD3232, VD3624
*R     10.0, VD3624
ROUND  VD3624, VD3624
Network 10
LDD<>  VD3624, VD1232
MOVD   VD3624, VD1232
DTI    VD3624, VW282
Network 11
LD     SM0.0
MOVR   VD3236, VD3628
*R     10.0, VD3628
ROUND  VD3628, VD3628
Network 12
LDD<>  VD3628, VD1236
MOVD   VD3628, VD1236
DTI    VD3628, VW284
Network 13
LD     SM0.0
MOVR   VD3244, VD3632
*R     10.0, VD3632
ROUND  VD3632, VD3632
Network 14
LDD<>  VD3632, VD1244
MOVD   VD3632, VD1244
DTI    VD3632, VW288
Network 15
LD     SM0.0
MOVR   VD3248, VD3636
*R     10.0, VD3636
ROUND  VD3636, VD3636
Network 16
LDD<>  VD3636, VD1248
MOVD   VD3636, VD1248
DTI    VD3636, VW290
Network 17
LD     SM0.0
MOVR   VD3252, VD3640
*R     10.0, VD3640
ROUND  VD3640, VD3640
Network 18
LDD<>  VD3640, VD1252
MOVD   VD3640, VD1252
DTI    VD3640, VW292
Network 19
LD     SM0.0
MOVR   VD3260, VD3644
*R     10.0, VD3644
ROUND  VD3644, VD3644
Network 20
LDD<>  VD3644, VD1260
MOVD   VD3644, VD1260
DTI    VD3644, VW296
Network 21
LD     SM0.0
MOVR   VD3000, VD3648
*R     100.0, VD3648
ROUND  VD3648, VD3648
Network 22
LDD<>  VD3648, VD2000
MOVD   VD3648, VD2000
DTI    VD3648, VW20
Network 23
LD     SM0.0
MOVR   VD3004, VD3652
*R     10.0, VD3652
ROUND  VD3652, VD3652
Network 24
LDD<>  VD3652, VD2004
MOVD   VD3652, VD2004
DTI    VD3652, VW24
Network 25
LD     SM0.0
MOVR   VD3008, VD3656
*R     10.0, VD3656
ROUND  VD3656, VD3656
Network 26
LDD<>  VD3656, VD2008
MOVD   VD3656, VD2008
DTI    VD3656, VW28
Network 27
LD     SM0.0
MOVR   VD3012, VD3660
*R     10.0, VD3660
ROUND  VD3660, VD3660
Network 28
LDD<>  VD3660, VD2012
MOVD   VD3660, VD2012
DTI    VD3660, VW32
Network 29
LD     SM0.0
MOVR   VD3016, VD3664
*R     10.0, VD3664
ROUND  VD3664, VD3664
Network 30
LDD<>  VD3664, VD2016
MOVD   VD3664, VD2016
DTI    VD3664, VW36
Network 31
LD     SM0.0
MOVR   VD3044, VD3672
*R     10.0, VD3672
ROUND  VD3672, VD3672
Network 32
LDD<>  VD3672, VD2044
MOVD   VD3672, VD2044
DTI    VD3672, VW44
Network 33
LD     SM0.0
MOVR   VD3048, VD3676
*R     10.0, VD3676
ROUND  VD3676, VD3676
Network 34
LDD<>  VD3676, VD2048
MOVD   VD3676, VD2048
DTI    VD3676, VW48
Network 35
LD     SM0.0
MOVR   VD3052, VD3680
*R     10.0, VD3680
ROUND  VD3680, VD3680
Network 36
LDD<>  VD3680, VD2052
MOVD   VD3680, VD2052
DTI    VD3680, VW52
Network 37
LD     SM0.0
MOVR   VD3056, VD3684
*R     10.0, VD3684
ROUND  VD3684, VD3684
Network 38
LDD<>  VD3684, VD2056
MOVD   VD3684, VD2056
DTI    VD3684, VW54
Network 39
LD     SM0.0
MOVR   VD3064, VD3688
*R     10.0, VD3688
ROUND  VD3688, VD3688
Network 40
LDD<>  VD3688, VD2064
MOVD   VD3688, VD2064
DTI    VD3688, VW58
Network 41
LD     SM0.0
MOVR   VD3082, VD3692
*R     10.0, VD3692
ROUND  VD3692, VD3692
Network 42
LDD<>  VD3692, VD2082
MOVD   VD3692, VD2082
DTI    VD3692, VW60
Network 43
LDW<>  VW3060, VW2060
MOVW   VW3060, VW2060
MOVW   VW3060, VW56
*I     +10, VW56
Network 44
LD     SM0.0
MOVR   VD3264, VD3668
*R     10.0, VD3668
ROUND  VD3668, VD3668
Network 45
LDD<>  VD3668, VD1264
MOVD   VD3668, VD1264
DTI    VD3668, VW298
Network 46
LD     SM0.0
MOVR   VD3130, VD3700
*R     10.0, VD3700
ROUND  VD3700, VD3700
Network 47
LDD<>  VD3700, VD2130
MOVD   VD3700, VD2130
DTI    VD3700, VW70
Network 48
LD     SM0.0
MOVR   VD3134, VD3704
*R     100.0, VD3704
ROUND  VD3704, VD3704
Network 49
LDD<>  VD3704, VD2134
MOVD   VD3704, VD2134
DTI    VD3704, VW72
Network 50
LD     SM0.0
MOVR   VD3138, VD3708
*R     10.0, VD3708
ROUND  VD3708, VD3708
Network 51
LDD<>  VD3708, VD2138
MOVD   VD3708, VD2138
DTI    VD3708, VW74
Network 52
LD     SM0.0
MOVR   VD3142, VD3712
*R     10.0, VD3712
ROUND  VD3712, VD3712
Network 53
LDD<>  VD3712, VD1178
MOVD   VD3712, VD1178
DTI    VD3712, VW76
Network 54
LD     SM0.0
MOVR   VD3150, VD3716
*R     10.0, VD3716
ROUND  VD3716, VD3716
Network 55
LDD<>  VD3716, VD2364
MOVD   VD3716, VD2364
DTI    VD3716, VW78
Network 56
LD     SM0.0
MOVR   VD3146, VD3696
*R     10.0, VD3696
ROUND  VD3696, VD3696
Network 57
LDD<>  VD3696, VD1174
MOVD   VD3696, VD1174
DTI    VD3696, VW300
END_SUBROUTINE_BLOCK

SUBROUTINE_BLOCK TOUCHER:SBR12
TITLE=
BEGIN
Network 1
LDN    M26.0
MOVB   0, VB742
Network 2
LD     M26.0
MOVB   10, VB742
Network 3
LDN    M26.4
MOVB   0, VB749
Network 4
LD     M26.4
MOVB   10, VB749
Network 5
LDN    M26.1
MOVB   0, VB751
Network 6
LD     M26.1
MOVB   10, VB751
Network 7
LD     M25.0
MOVD   VD4070, VD3070
MOVD   VD4074, VD3074
MOVD   VD4078, VD3078
MOVD   VD4086, VD3086
MOVD   VD4090, VD3090
MOVD   VD4094, VD3094
BMW    VW4500, VW2200, 5
BMW    VW4512, VW2212, 5
MOVW   VW4660, VW2360
MOVW   VW4662, VW2362
Network 8
LD     M25.0
MOVD   VD4102, VD3102
MOVD   VD4106, VD3106
MOVD   VD4110, VD3110
MOVD   VD4118, VD3118
MOVD   VD4122, VD3122
MOVD   VD4126, VD3126
BMW    VW4524, VW2224, 5
BMW    VW4536, VW2236, 5
Network 9
LD     M25.0
MOVD   VD4196, VD3196
MOVD   VD4200, VD3200
MOVD   VD4204, VD3204
MOVD   VD4212, VD3212
MOVD   VD4216, VD3216
MOVD   VD4220, VD3220
BMW    VW4596, VW2296, 5
BMW    VW4608, VW2308, 5
Network 10
LD     M25.0
MOVD   VD4228, VD3228
MOVD   VD4232, VD3232
MOVD   VD4236, VD3236
MOVD   VD4244, VD3244
MOVD   VD4248, VD3248
MOVD   VD4252, VD3252
BMW    VW4620, VW2320, 5
BMW    VW4632, VW2332, 5
R      M25.0, 1
Network 11
LD     M25.1
MOVD   VD4004, VD3004
MOVD   VD4008, VD3008
MOVD   VD4012, VD3012
MOVD   VD4000, VD3000
MOVD   VD4052, VD3052
MOVD   VD4020, VD3130
R      M25.1, 1
Network 12
LD     M25.2
MOVD   VD4016, VD3016
MOVD   VD4044, VD3044
MOVD   VD4048, VD3048
MOVD   VD4264, VD3264
MOVD   VD4024, VD3134
R      M25.2, 1
Network 13
LD     M25.3
MOVD   VD4260, VD3260
BMW    VW4644, VW2344, 2
BMW    VW4650, VW2350, 5
MOVD   VD4028, VD3142
MOVD   VD4032, VD3146
MOVD   VD4036, VD3150
R      M25.3, 1
Network 14
LDW<>  VW1274, VW736
MOVW   VW1274, VW736
Network 15
LD     M31.7
LPS
AD<>   VD10, +369
AD<>   VD10, +8410
AD<>   VD10, +2140
S      M31.3, 1
LPP
AD=    VD10, +369
S      M31.1, 1
R      M31.2, 1
R      M31.3, 1
S      M31.4, 1
MOVD   +0, VD10
Network 16
LDN    M31.7
R      M31.3, 1
Network 17
LD     M31.7
AD=    VD10, +8410
S      M31.2, 1
R      M31.1, 1
R      M31.3, 1
S      M31.4, 1
MOVD   +0, VD10
Network 18
LD     M31.7
AD=    VD10, +2140
R      M31.1, 3
S      M31.4, 1
R      M31.0, 1
MOVD   +0, VD10
Network 19
LD     M26.6
CALL   Load_Data:SBR21
CALL   Init_Public_Var:SBR14
R      M26.6, 1
Network 20
LD     M26.5
CALL   Save_Data:SBR20
R      M26.5, 1
Network 21
LDW<>  VW1000, VW82
MOVW   VW1000, VW82
Network 22
LDW<>  VW1002, VW86
MOVW   VW1002, VW86
Network 23
LDW<>  VW1004, VW90
MOVW   VW1004, VW90
Network 24
LDW<>  VW1008, VW148
MOVW   VW1008, VW148
Network 25
LDW<>  VW1010, VW152
MOVW   VW1010, VW152
Network 26
LDW<>  VW1012, VW804
MOVW   VW1012, VW804
Network 27
LDW<>  VW1014, VW808
MOVW   VW1014, VW808
Network 28
LDW<>  VW1016, VW814
MOVW   VW1016, VW814
Network 29
LDW<>  VW1020, VW824
MOVW   VW1020, VW824
Network 30
LDW<>  VW2200, VW380
MOVW   VW2200, VW380
Network 31
LDW<>  VW2202, VW382
MOVW   VW2202, VW382
Network 32
LDW<>  VW2204, VW384
MOVW   VW2204, VW384
Network 33
LDW<>  VW2206, VW386
MOVW   VW2206, VW386
Network 34
LDW<>  VW2208, VW388
MOVW   VW2208, VW388
Network 35
LDW<>  VW2212, VW392
MOVW   VW2212, VW392
Network 36
LDW<>  VW2214, VW394
MOVW   VW2214, VW394
Network 37
LDW<>  VW2216, VW396
MOVW   VW2216, VW396
Network 38
LDW<>  VW2218, VW398
MOVW   VW2218, VW398
Network 39
LDW<>  VW2220, VW400
MOVW   VW2220, VW400
Network 40
LDW<>  VW2224, VW404
MOVW   VW2224, VW404
Network 41
LDW<>  VW2226, VW406
MOVW   VW2226, VW406
Network 42
LDW<>  VW2228, VW408
MOVW   VW2228, VW408
Network 43
LDW<>  VW2230, VW410
MOVW   VW2230, VW410
Network 44
LDW<>  VW2232, VW412
MOVW   VW2232, VW412
Network 45
LDW<>  VW2236, VW416
MOVW   VW2236, VW416
Network 46
LDW<>  VW2238, VW418
MOVW   VW2238, VW418
Network 47
LDW<>  VW2240, VW420
MOVW   VW2240, VW420
Network 48
LDW<>  VW2242, VW422
MOVW   VW2242, VW422
Network 49
LDW<>  VW2244, VW424
MOVW   VW2244, VW424
Network 50
LDW<>  VW2296, VW476
MOVW   VW2296, VW476
Network 51
LDW<>  VW2298, VW478
MOVW   VW2298, VW478
Network 52
LDW<>  VW2300, VW480
MOVW   VW2300, VW480
Network 53
LDW<>  VW2302, VW482
MOVW   VW2302, VW482
Network 54
LDW<>  VW2304, VW484
MOVW   VW2304, VW484
Network 55
LDW<>  VW2308, VW488
MOVW   VW2308, VW488
Network 56
LDW<>  VW2310, VW490
MOVW   VW2310, VW490
Network 57
LDW<>  VW2312, VW492
MOVW   VW2312, VW492
Network 58
LDW<>  VW2314, VW494
MOVW   VW2314, VW494
Network 59
LDW<>  VW2316, VW496
MOVW   VW2316, VW496
Network 60
LDW<>  VW2320, VW500
MOVW   VW2320, VW500
Network 61
LDW<>  VW2322, VW502
MOVW   VW2322, VW502
Network 62
LDW<>  VW2324, VW504
MOVW   VW2324, VW504
Network 63
LDW<>  VW2326, VW506
MOVW   VW2326, VW506
Network 64
LDW<>  VW2328, VW508
MOVW   VW2328, VW508
Network 65
LDW<>  VW2332, VW512
MOVW   VW2332, VW512
Network 66
LDW<>  VW2334, VW514
MOVW   VW2334, VW514
Network 67
LDW<>  VW2336, VW516
MOVW   VW2336, VW516
Network 68
LDW<>  VW2338, VW518
MOVW   VW2338, VW518
Network 69
LDW<>  VW2340, VW520
MOVW   VW2340, VW520
Network 70
LDW<>  VW2344, VW524
MOVW   VW2344, VW524
Network 71
LDW<>  VW2346, VW526
MOVW   VW2346, VW526
Network 72
LDW<>  VW2350, VW530
MOVW   VW2350, VW530
Network 73
LDW<>  VW2352, VW532
MOVW   VW2352, VW532
Network 74
LDW<>  VW2354, VW534
MOVW   VW2354, VW534
Network 75
LDW<>  VW2356, VW536
MOVW   VW2356, VW536
Network 76
LDW<>  VW2358, VW538
MOVW   VW2358, VW538
END_SUBROUTINE_BLOCK

SUBROUTINE_BLOCK SYSRESET:SBR13
TITLE=
BEGIN
Network 1
LD     SM0.0
CALL   RESET:SBR2
CALL   RESET1:SBR9
Network 2
LD     SM0.0
CALL   Init_Public_Var:SBR14
Network 3
LD     SM0.0
BTI    VB2450, VW5162
MOVW   VW5162, VW5130
BCDI   VW5130
Network 4
LD     SM0.0
BTI    VB2451, VW5164
MOVW   VW5164, VW5132
BCDI   VW5132
Network 5
LD     SM0.0
BTI    VB2452, VW5166
MOVW   VW5166, VW5134
BCDI   VW5134
Network 6
LD     SM0.0
BTI    VB2453, VW5168
MOVW   VW5168, VW5136
BCDI   VW5136
Network 7
LD     SM0.0
BTI    VB2454, VW5170
MOVW   VW5170, VW5138
BCDI   VW5138
Network 8
LD     SM0.0
BTI    VB2455, VW5172
MOVW   VW5172, VW5140
BCDI   VW5140
Network 9
LD     SM0.0
R      M26.0, 2
R      M26.4, 1
Network 10
LD     SM0.0
R      M3.1, 1
S      M3.0, 1
R      M3.3, 1
R      M31.7, 1
R      M31.1, 2
R      M31.4, 1
S      M31.0, 1
R      M31.6, 1
MOVD   +0, VD10
Network 11
LD     SM0.0
MOVW   VW1000, VW82
MOVW   VW1002, VW86
MOVW   VW1006, VW94
MOVW   VW1004, VW90
Network 12
LD     SM0.0
MOVW   VW1012, VW804
MOVW   VW1014, VW808
Network 13
LD     SM0.0
MOVW   VW1274, VW736
MOVW   VW1016, VW814
Network 14
LD     SM0.0
MOVW   VW1020, VW824
END_SUBROUTINE_BLOCK

SUBROUTINE_BLOCK Init_Public_Var:SBR14
TITLE=
BEGIN
Network 1
LD     SM0.0
BMW    VW2350, VW530, 5
MOVW   VW2360, VW540
MOVW   VW2362, VW542
Network 2
LD     SM0.0
DTI    VD2130, VW70
DTR    VD2130, VD3700
AENO
MOVR   VD3700, VD3130
/R     10.0, VD3130
Network 3
LD     SM0.0
DTI    VD2134, VW72
DTR    VD2134, VD3704
AENO
MOVR   VD3704, VD3134
/R     100.0, VD3134
Network 4
LD     SM0.0
DTI    VD2138, VW74
DTR    VD2138, VD3708
AENO
MOVR   VD3708, VD3138
/R     10.0, VD3138
Network 5
LD     SM0.0
DTI    VD1178, VW76
DTR    VD1178, VD3712
AENO
MOVR   VD3712, VD3142
/R     10.0, VD3142
Network 6
LD     SM0.0
DTI    VD1174, VW300
DTR    VD1174, VD3696
AENO
MOVR   VD3696, VD3146
/R     10.0, VD3146
Network 7
LD     SM0.0
DTI    VD2364, VW78
DTR    VD2364, VD3716
AENO
MOVR   VD3716, VD3150
/R     10.0, VD3150
Network 8
LD     SM0.0
MOVW   VW1008, VW148
MOVW   VW1010, VW152
Network 9
LD     SM0.0
BMW    VW2200, VW380, 5
BMW    VW2212, VW392, 5
Network 10
LD     SM0.0
BMW    VW2224, VW404, 5
BMW    VW2236, VW416, 5
Network 11
LD     SM0.0
BMW    VW2296, VW476, 5
BMW    VW2308, VW488, 5
Network 12
LD     SM0.0
BMW    VW2320, VW500, 5
BMW    VW2332, VW512, 5
MOVW   VW2344, VW524
MOVW   VW2346, VW526
Network 13
LD     SM0.0
DTI    VD2070, VW200
DTR    VD2070, VD3500
AENO
MOVR   VD3500, VD3070
/R     10.0, VD3070
Network 14
LD     SM0.0
DTI    VD2074, VW202
DTR    VD2074, VD3504
AENO
MOVR   VD3504, VD3074
/R     10.0, VD3074
Network 15
LD     SM0.0
DTI    VD2078, VW204
DTR    VD2078, VD3508
AENO
MOVR   VD3508, VD3078
/R     10.0, VD3078
Network 16
LD     SM0.0
DTI    VD2086, VW208
DTR    VD2086, VD3512
AENO
MOVR   VD3512, VD3086
/R     10.0, VD3086
Network 17
LD     SM0.0
DTI    VD2090, VW210
DTR    VD2090, VD3516
AENO
MOVR   VD3516, VD3090
/R     10.0, VD3090
Network 18
LD     SM0.0
DTI    VD2094, VW212
DTR    VD2094, VD3520
AENO
MOVR   VD3520, VD3094
/R     10.0, VD3094
Network 19
LD     SM0.0
DTI    VD2102, VW216
DTR    VD2102, VD3524
AENO
MOVR   VD3524, VD3102
/R     10.0, VD3102
Network 20
LD     SM0.0
DTI    VD2106, VW218
DTR    VD2106, VD3528
AENO
MOVR   VD3528, VD3106
/R     10.0, VD3106
Network 21
LD     SM0.0
DTI    VD2110, VW220
DTR    VD2110, VD3532
AENO
MOVR   VD3532, VD3110
/R     10.0, VD3110
Network 22
LD     SM0.0
DTI    VD2118, VW224
DTR    VD2118, VD3536
AENO
MOVR   VD3536, VD3118
/R     10.0, VD3118
Network 23
LD     SM0.0
DTI    VD2122, VW226
DTR    VD2122, VD3540
AENO
MOVR   VD3540, VD3122
/R     10.0, VD3122
Network 24
LD     SM0.0
DTI    VD2126, VW228
DTR    VD2126, VD3544
AENO
MOVR   VD3544, VD3126
/R     10.0, VD3126
Network 25
LD     SM0.0
DTI    VD1196, VW264
DTR    VD1196, VD3596
AENO
MOVR   VD3596, VD3196
/R     10.0, VD3196
Network 26
LD     SM0.0
DTI    VD1200, VW266
DTR    VD1200, VD3600
AENO
MOVR   VD3600, VD3200
/R     10.0, VD3200
Network 27
LD     SM0.0
DTI    VD1204, VW268
DTR    VD1204, VD3604
AENO
MOVR   VD3604, VD3204
/R     10.0, VD3204
Network 28
LD     SM0.0
DTI    VD1212, VW272
DTR    VD1212, VD3608
AENO
MOVR   VD3608, VD3212
/R     10.0, VD3212
Network 29
LD     SM0.0
DTI    VD1216, VW274
DTR    VD1216, VD3612
AENO
MOVR   VD3612, VD3216
/R     10.0, VD3216
Network 30
LD     SM0.0
DTI    VD1220, VW276
DTR    VD1220, VD3616
AENO
MOVR   VD3616, VD3220
/R     10.0, VD3220
Network 31
LD     SM0.0
DTI    VD1228, VW280
DTR    VD1228, VD3620
AENO
MOVR   VD3620, VD3228
/R     10.0, VD3228
Network 32
LD     SM0.0
DTI    VD1232, VW282
DTR    VD1232, VD3624
AENO
MOVR   VD3624, VD3232
/R     10.0, VD3232
Network 33
LD     SM0.0
DTI    VD1236, VW284
DTR    VD1236, VD3628
AENO
MOVR   VD3628, VD3236
/R     10.0, VD3236
Network 34
LD     SM0.0
DTI    VD1244, VW288
DTR    VD1244, VD3632
AENO
MOVR   VD3632, VD3244
/R     10.0, VD3244
Network 35
LD     SM0.0
DTI    VD1248, VW290
DTR    VD1248, VD3636
AENO
MOVR   VD3636, VD3248
/R     10.0, VD3248
Network 36
LD     SM0.0
DTI    VD1252, VW292
DTR    VD1252, VD3640
AENO
MOVR   VD3640, VD3252
/R     10.0, VD3252
Network 37
LD     SM0.0
DTI    VD1260, VW296
DTR    VD1260, VD3644
AENO
MOVR   VD3644, VD3260
/R     10.0, VD3260
Network 38
LD     SM0.0
DTI    VD2000, VW20
DTR    VD2000, VD3648
AENO
MOVR   VD3648, VD3000
/R     100.0, VD3000
Network 39
LD     SM0.0
DTI    VD2004, VW24
DTR    VD2004, VD3652
AENO
MOVR   VD3652, VD3004
/R     10.0, VD3004
Network 40
LD     SM0.0
DTI    VD2008, VW28
DTR    VD2008, VD3656
AENO
MOVR   VD3656, VD3008
/R     10.0, VD3008
Network 41
LD     SM0.0
DTI    VD2012, VW32
DTR    VD2012, VD3660
AENO
MOVR   VD3660, VD3012
/R     10.0, VD3012
Network 42
LD     SM0.0
DTI    VD2016, VW36
DTR    VD2016, VD3664
AENO
MOVR   VD3664, VD3016
/R     10.0, VD3016
Network 43
LD     SM0.0
DTI    VD2044, VW44
DTR    VD2044, VD3672
AENO
MOVR   VD3672, VD3044
/R     10.0, VD3044
Network 44
LD     SM0.0
DTI    VD2048, VW48
DTR    VD2048, VD3676
AENO
MOVR   VD3676, VD3048
/R     10.0, VD3048
Network 45
LD     SM0.0
DTI    VD2052, VW52
DTR    VD2052, VD3680
AENO
MOVR   VD3680, VD3052
/R     10.0, VD3052
Network 46
LD     SM0.0
DTI    VD2056, VW54
DTR    VD2056, VD3684
AENO
MOVR   VD3684, VD3056
/R     10.0, VD3056
Network 47
LD     SM0.0
DTI    VD2064, VW58
DTR    VD2064, VD3688
AENO
MOVR   VD3688, VD3064
/R     10.0, VD3064
Network 48
LD     SM0.0
DTI    VD2082, VW60
DTR    VD2082, VD3692
AENO
MOVR   VD3692, VD3082
/R     10.0, VD3082
Network 49
LD     SM0.0
MOVW   VW2060, VW3060
MOVW   VW2060, VW56
*I     +10, VW56
Network 50
LD     SM0.0
DTI    VD1264, VW298
DTR    VD1264, VD3668
AENO
MOVR   VD3668, VD3264
/R     10.0, VD3264
END_SUBROUTINE_BLOCK

SUBROUTINE_BLOCK AUTO_PRODUCT:SBR15
TITLE=
BEGIN
Network 1
LDN    M29.3
A      M29.1
S      M12.5, 1
TON    T99, VW20
A      T99
R      T99, 1
R      M12.5, 1
R      T156, 1
S      M29.3, 1
Network 2
LD     M29.3
TON    T156, VW70
A      T156
R      T156, 1
R      M29.1, 1
R      M29.3, 1
R      M28.7, 1
Network 3
LDB=   VB700, 100
LD     I0.3
O      M22.1
ALD
AW>=   VW804, +1
AN     M3.3
A      I2.5
A      I2.6
A      I3.1
A      I3.3
MOVB   58, VB700
MOVW   +0, VW802
MOVW   +0, VW806
MOVB   100, VB702
Network 4
LDB=   VB700, 58
LD     I0.3
O      M22.1
ALD
AW>=   VW804, +1
AN     M3.3
A      I2.5
A      I2.6
A      I3.1
A      I3.3
S      M3.1, 1
R      M3.0, 1
S      Q1.7, 1
MOVB   56, VB700
Network 5
LDB=   VB700, 56
LPS
A      I3.2
S      M10.1, 1
LRD
R      T162, 1
LRD
A      I3.2
MOVB   55, VB700
LPP
AN     I3.2
MOVB   54, VB700
Network 6
LDB=   VB700, 55
TON    T162, VW28
A      T162
R      M10.1, 1
R      T162, 1
MOVB   54, VB700
Network 7
LDB=   VB700, 54
AN     M3.3
MOVB   52, VB700
Network 8
LDB=   VB700, 52
CALL   CLOTH_PROCESS:SBR16
Network 9
LDB=   VB700, 48
R      T110, 1
MOVB   46, VB700
Network 10
LDB=   VB700, 46
S      M10.1, 1
TON    T110, VW28
A      T110
R      M10.1, 1
R      T110, 1
MOVB   44, VB700
Network 11
LDB=   VB700, 44
AN     V5005.0
AN     I2.5
TON    T203, +8
A      T203
R      T203, 1
S      V5005.0, 1
R      M11.6, 1
Network 12
LDB=   VB700, 44
A      I2.5
S      M11.6, 1
R      T116, 1
MOVB   43, VB700
Network 13
LDB=   VB700, 43
TON    T116, VW48
A      T116
R      T116, 1
R      V5005.0, 1
R      M11.6, 1
MOVB   42, VB700
Network 14
LDB=   VB700, 42
S      M12.0, 1
S      Q1.3, 1
MOVB   40, VB700
Network 15
LDB=   VB700, 40
A      I2.7
AB=    VB749, 10
R      T129, 1
R      T127, 1
Network 16
LDB=   VB700, 40
A      I2.7
R      M12.0, 1
R      Q1.3, 1
MOVB   36, VB700
Network 17
LDB=   VB700, 40
A      Q1.3
TON    T148, VW298
A      T148
R      T148, 1
R      Q1.3, 1
Network 18
LDB=   VB700, 40
AB=    VB749, 10
TON    T127, VW300
A      T127
R      T127, 1
R      M12.0, 1
R      Q1.3, 1
R      T129, 1
MOVB   110, VB700
Network 19
LDB=   VB700, 110
S      M11.4, 1
TON    T129, VW76
A      T129
R      T129, 1
R      M11.4, 1
MOVB   108, VB700
Network 20
LDB=   VB700, 108
S      M12.0, 1
S      Q1.3, 1
MOVB   106, VB700
Network 21
LDB=   VB700, 106
A      I2.7
R      M12.0, 1
R      Q1.3, 1
MOVB   36, VB700
Network 22
LDB=   VB700, 36
TON    T122, VW32
A      T122
R      T122, 1
R      T100, 1
MOVB   35, VB700
Network 23
LDB=   VB700, 35
S      M11.4, 1
TON    T100, VW72
A      T100
R      T100, 1
R      M11.4, 1
MOVB   34, VB700
Network 24
LDB=   VB700, 34
AN     I2.5
AN     V5003.1
TON    T204, +8
A      T204
R      T204, 1
S      V5003.1, 1
R      M30.0, 1
Network 25
LDB=   VB700, 34
LPS
A      I2.5
S      M30.0, 1
LPP
A      I3.0
MOVB   32, VB700
Network 26
LDB=   VB700, 32
TON    T36, +5
A      T36
LPS
R      T36, 1
A      I3.0
R      M30.0, 1
R      V5003.1, 1
MOVB   30, VB700
INCW   VW802
INCD   VD1190
LPP
AN     I3.0
MOVB   34, VB700
Network 27
LDB=   VB700, 30
LPS
S      M11.4, 1
A      I3.3
S      M18.7, 1
LRD
AN     I3.3
S      V5005.5, 1
S      M30.7, 1
LPP
MOVB   28, VB700
Network 28
LDB=   VB700, 28
AN     I4.1
AN     M21.6
AN     Q1.5
A      I3.3
S      M21.6, 1
R      M18.7, 1
S      M30.4, 1
S      Q1.5, 1
MOVB   27, VB700
Network 29
LDB=   VB700, 28
A      Q1.5
MOVB   27, VB700
Network 30
LDB=   VB700, 28
OB=    VB700, 27
A      I2.6
MOVB   26, VB700
Network 31
LDB=   VB700, 26
TON    T98, +5
A      T98
LPS
R      T98, 1
A      I2.6
R      M11.4, 1
MOVB   24, VB700
LPP
AN     I2.6
MOVB   27, VB700
Network 32
LDB=   VB700, 24
AN     M29.7
AN     I4.1
AN     Q1.5
AN     M21.6
S      M21.6, 1
R      M18.7, 1
S      M30.4, 1
S      Q1.5, 1
MOVB   23, VB700
Network 33
LDB=   VB700, 24
OB=    VB700, 23
A      M29.7
S      M12.3, 1
A      I3.1
MOVB   22, VB700
Network 34
LDB=   VB700, 22
TON    T97, +5
A      T97
LPS
R      T97, 1
A      I3.1
R      M29.7, 1
R      M12.3, 1
MOVB   20, VB700
LPP
AN     I3.1
MOVB   23, VB700
Network 35
LDB=   VB700, 20
AW<    VW802, VW804
MOVB   54, VB700
Network 36
LDB=   VB700, 20
AW=    VW802, VW804
R      M3.1, 1
S      M3.0, 1
S      M28.6, 1
R      Q1.7, 1
MOVB   100, VB700
END_SUBROUTINE_BLOCK

SUBROUTINE_BLOCK CLOTH_PROCESS:SBR16
TITLE=
BEGIN
Network 1
LDN    M29.0
A      I2.4
TON    T33, +5
A      T33
R      T33, 1
S      M29.0, 1
Network 2
LD     SM0.0
LPS
AN     I2.4
R      M29.0, 1
LPP
A      M29.0
EU
INCW   VW806
AW=    VW806, VW736
AN     M29.1
AN     M29.2
S      M29.1, 1
S      M29.2, 1
R      T99, 1
R      M29.3, 1
Network 3
LD     M29.4
TON    T114, VW24
A      T114
R      T114, 1
S      M29.5, 1
R      M29.4, 1
Network 4
LD     M29.5
S      Q0.2, 1
A      I3.2
R      M29.5, 1
S      M29.6, 1
Network 5
LD     M29.6
TON    T34, +5
A      T34
LPS
R      T34, 1
A      I3.2
R      Q0.2, 1
R      M29.4, 3
LPP
AN     I3.2
S      M29.5, 1
Network 6
LDB=   VB702, 100
LPS
S      M18.1, 1
AN     I3.2
S      M29.4, 1
LPP
A      I2.4
MOVB   90, VB702
Network 7
LDB=   VB702, 90
A      M29.0
S      Q1.4, 1
R      M18.1, 1
AW<    VW806, VW808
MOVB   85, VB702
Network 8
LDB=   VB702, 90
A      M29.0
AW>=   VW806, VW808
LPS
AB=    VB751, 0
MOVB   60, VB702
LPP
AB=    VB751, 10
MOVB   72, VB702
Network 9
LDB=   VB702, 85
LD     M29.2
AN     M29.1
ON     M29.2
ALD
S      M18.4, 1
MOVB   80, VB702
Network 10
LDB=   VB702, 80
TON    T124, VW52
A      T124
R      T124, 1
R      M18.4, 1
MOVB   78, VB702
Network 11
LDB=   VB702, 78
S      M18.1, 1
A      I2.4
MOVB   76, VB702
Network 12
LDB=   VB702, 76
A      M29.0
S      Q1.4, 1
R      M18.1, 1
AW<    VW806, VW808
MOVB   85, VB702
Network 13
LDB=   VB702, 76
A      M29.0
AW>=   VW806, VW808
LPS
AB=    VB751, 0
MOVB   60, VB702
LPP
AB=    VB751, 10
MOVB   72, VB702
Network 14
LDB=   VB702, 72
LD     M29.2
AN     M29.1
ON     M29.2
ALD
R      Q1.4, 1
A      I2.6
S      M18.4, 1
Network 15
LDB=   VB702, 72
A      I2.5
MOVB   70, VB702
Network 16
LDB=   VB702, 70
TON    T187, +1
A      T187
LPS
R      T187, 1
A      I2.5
R      M18.4, 1
R      T164, 1
MOVB   68, VB702
LPP
AN     I2.5
MOVB   72, VB702
Network 17
LDB=   VB702, 68
S      M10.1, 1
TON    T164, VW28
A      T164
R      M10.1, 1
R      T164, 1
R      T131, 1
MOVB   67, VB702
Network 18
LDB=   VB702, 67
TON    T131, VW78
A      T131
R      T131, 1
MOVB   66, VB702
Network 19
LDB=   VB702, 66
S      M10.0, 1
A      I3.2
R      M10.0, 1
MOVB   64, VB702
Network 20
LDB=   VB702, 64
LPS
A      I2.6
S      M18.1, 1
LPP
A      I2.4
MOVB   63, VB702
Network 21
LDB=   VB702, 63
A      M29.0
S      Q1.4, 1
R      M18.1, 1
R      T158, 1
MOVB   62, VB702
Network 22
LDB=   VB702, 62
TON    T158, VW70
A      T158
R      T158, 1
MOVB   60, VB702
Network 23
LDB=   VB702, 60
LD     M29.2
AN     M29.1
ON     M29.2
ALD
S      M18.4, 1
R      M29.2, 1
R      Q1.4, 1
MOVB   55, VB702
Network 24
LDB=   VB702, 55
A      I2.5
MOVB   53, VB702
Network 25
LDB=   VB702, 53
TON    T35, +5
A      T35
LPS
R      T35, 1
A      I2.5
R      M18.4, 1
MOVB   50, VB702
LPP
AN     I2.5
MOVB   55, VB702
Network 26
LDB=   VB702, 50
MOVW   +0, VW806
MOVB   48, VB700
MOVB   100, VB702
END_SUBROUTINE_BLOCK

SUBROUTINE_BLOCK Manual_Spot:SBR17
TITLE=
BEGIN
Network 1
LDN    M2.0
AB=    VB742, 10
LD     I1.6
O      M23.4
ALD
S      M2.0, 1
S      M18.0, 1
S      Q1.5, 1
Network 2
LD     M2.0
A      Q1.5
AN     I3.3
AN     M2.1
S      M2.1, 1
Network 3
LD     M2.0
A      M2.1
A      I3.3
R      M2.0, 2
R      M18.0, 1
R      Q1.5, 1
Network 4
LD     M2.0
LDN    M23.4
AN     I1.6
OB=    VB742, 0
ALD
R      M18.0, 1
R      M2.0, 2
R      M18.5, 1
R      Q1.5, 1
Network 5
LD     M7.6
A      Q1.3
LD     I2.0
O      M23.6
ALD
ED
R      M12.5, 1
R      M7.6, 1
Network 6
LD     M12.5
AN     M12.7
TON    T99, VW20
A      T99
R      T99, 1
S      M12.7, 1
Network 7
LD     M7.6
A      Q1.3
A      M12.7
R      M12.5, 1
R      M7.6, 1
Network 8
LDN    M7.6
AN     M12.7
LD     I2.0
O      M23.6
ALD
ED
S      M7.6, 1
S      M12.5, 1
Network 9
LD     M7.7
AB=    VB742, 0
A      Q1.5
LD     I1.6
O      M23.4
ALD
ED
R      M18.0, 1
R      M7.7, 1
R      M2.2, 1
R      Q1.5, 1
Network 10
LD     M7.7
A      Q1.5
AN     I3.3
AN     M2.2
S      M2.2, 1
Network 11
LD     M7.7
A      M2.2
A      I3.3
R      M18.0, 1
R      M7.7, 1
R      M2.2, 1
R      Q1.5, 1
Network 12
LD     M7.7
A      Q1.5
LDB=   VB742, 10
ON     I3.0
O      I2.2
ALD
R      M18.0, 1
R      M7.7, 1
R      M2.2, 1
R      Q1.5, 1
Network 13
LDN    M7.7
AB=    VB742, 0
A      I3.0
LD     I1.6
O      M23.4
ALD
ED
S      M7.7, 1
S      M18.0, 1
S      Q1.5, 1
Network 14
LDN    M18.2
LD     I1.7
O      M23.5
ALD
ED
S      M18.2, 1
S      Q1.6, 1
Network 15
LD     M18.2
A      Q1.6
LD     I1.7
O      M23.5
ALD
ED
R      M18.2, 1
R      Q1.6, 1
R      M2.3, 1
Network 16
LD     M18.2
A      Q1.6
LD     I4.1
O      M2.3
ALD
R      M18.2, 1
R      Q1.6, 1
R      M2.3, 1
Network 17
LDN    M18.3
LD     I2.1
O      M23.7
ALD
ED
S      M18.3, 1
S      Q1.4, 1
Network 18
LD     M18.3
A      Q1.4
LD     I2.1
O      M23.7
ALD
ED
R      M18.3, 1
R      Q1.4, 1
Network 19
LDN    M4.3
A      M4.2
TON    T163, VW28
A      T163
R      M10.1, 1
R      T163, 1
R      M4.2, 1
S      M4.3, 1
Network 20
LDN    M4.6
A      M4.3
TON    T168, VW78
A      T168
R      T168, 1
S      M4.6, 1
Network 21
LD     M4.6
S      M10.0, 1
LD     I3.2
O      M8.1
ALD
R      M10.0, 1
R      M4.3, 1
R      M4.6, 1
END_SUBROUTINE_BLOCK

SUBROUTINE_BLOCK Trou_Run:SBR18
TITLE=
BEGIN
Network 1
LD     M4.1
AN     I2.3
=      V5000.0
Network 2
LD     I2.2
=      V5000.1
Network 3
LD     I1.6
O      M23.4
AN     I3.0
AN     V5002.0
AB=    VB742, 0
=      V5002.0
Network 4
LD     Q1.6
AN     M2.3
TON    T120, VW44
A      T120
R      T120, 1
S      M2.3, 1
S      V5003.2, 1
Network 5
LD     V5003.2
TON    T182, +6
A      T182
R      T182, 1
R      V5003.2, 1
Network 6
LD     M12.5
LDN    I0.0
A      M12.0
OLD
S      Q1.3, 1
Network 7
LDN    M12.5
LPS
AN     M12.0
R      Q1.3, 1
LPP
R      M12.7, 1
Network 8
LD     M12.0
AN     M12.6
TON    T128, VW296
A      T128
R      T128, 1
S      M12.6, 1
S      V5002.6, 1
Network 9
LD     V5002.6
TON    T183, +6
A      T183
R      T183, 1
R      V5002.6, 1
Network 10
LDN    M12.0
R      M12.6, 1
Network 11
LD     M1.4
OB=    VB701, 80
AN     M9.4
TON    T152, VW56
A      T152
R      T152, 1
S      M9.4, 1
S      V5005.7, 1
END_SUBROUTINE_BLOCK

SUBROUTINE_BLOCK SETUP_DATE:SBR19
TITLE=
BEGIN
Network 1
LD     M26.3
MOVW   VW5130, VW5150
IBCD   VW5150
ITB    VW5150, VB5120
Network 2
LD     M26.3
MOVW   VW5132, VW5152
IBCD   VW5152
ITB    VW5152, VB5121
Network 3
LD     M26.3
MOVW   VW5134, VW5154
IBCD   VW5154
ITB    VW5154, VB5122
Network 4
LD     M26.3
MOVW   VW5136, VW5156
IBCD   VW5156
ITB    VW5156, VB5123
Network 5
LD     M26.3
MOVW   VW5138, VW5158
IBCD   VW5158
ITB    VW5158, VB5124
Network 6
LD     M26.3
MOVW   VW5140, VW5160
IBCD   VW5160
ITB    VW5160, VB5125
MOVB   0, VB5126
Network 7
LD     M26.3
TODW   VB5120
R      M26.3, 1
END_SUBROUTINE_BLOCK

SUBROUTINE_BLOCK Save_Data:SBR20
TITLE=
BEGIN
Network 1
LD     SM0.0
BMW    VW1008, VW2500, 2
BMD    VD1174, VD2504, 2
BMD    VD1196, VD2520, 3
BMD    VD1212, VD2532, 3
Network 2
LD     SM0.0
BMD    VD1228, VD2544, 3
BMD    VD1244, VD2556, 3
BMD    VD1260, VD2568, 2
BMD    VD2000, VD2576, 5
BMD    VD2044, VD2596, 3
Network 3
LD     SM0.0
BMD    VD2070, VD2608, 3
BMD    VD2086, VD2620, 3
BMD    VD2102, VD2632, 3
BMD    VD2118, VD2644, 4
Network 4
LD     SM0.0
BMW    VW2200, VW2660, 5
BMW    VW2212, VW2672, 5
BMW    VW2224, VW2684, 5
BMW    VW2236, VW2696, 5
BMW    VW2296, VW2708, 5
Network 5
LD     SM0.0
BMW    VW2308, VW2720, 5
BMW    VW2320, VW2732, 5
BMW    VW2332, VW2744, 5
BMW    VW2344, VW2756, 2
BMW    VW2350, VW2762, 5
BMW    VW2360, VW2772, 2
Network 6
LD     SM0.0
MOVD   VD2364, VD2776
BMD    VD2134, VD2780, 2
BMD    VD2056, VD2788, 3
MOVD   VD2082, VD2516
END_SUBROUTINE_BLOCK

SUBROUTINE_BLOCK Load_Data:SBR21
TITLE=
BEGIN
Network 1
LD     SM0.0
BMW    VW2500, VW1008, 2
BMD    VD2504, VD1174, 2
BMD    VD2520, VD1196, 3
BMD    VD2532, VD1212, 3
Network 2
LD     SM0.0
BMD    VD2544, VD1228, 3
BMD    VD2556, VD1244, 3
BMD    VD2568, VD1260, 2
BMD    VD2576, VD2000, 5
BMD    VD2596, VD2044, 3
Network 3
LD     SM0.0
BMD    VD2608, VD2070, 3
BMD    VD2620, VD2086, 3
BMD    VD2632, VD2102, 3
BMD    VD2644, VD2118, 4
Network 4
LD     SM0.0
BMW    VW2660, VW2200, 5
BMW    VW2672, VW2212, 5
BMW    VW2684, VW2224, 5
BMW    VW2696, VW2236, 5
BMW    VW2708, VW2296, 5
Network 5
LD     SM0.0
BMW    VW2720, VW2308, 5
BMW    VW2732, VW2320, 5
BMW    VW2744, VW2332, 5
BMW    VW2756, VW2344, 2
BMW    VW2762, VW2350, 5
BMW    VW2772, VW2360, 2
Network 6
LD     SM0.0
MOVD   VD2776, VD2364
BMD    VD2780, VD2134, 2
BMD    VD2788, VD2056, 3
MOVD   VD2516, VD2082
END_SUBROUTINE_BLOCK

SUBROUTINE_BLOCK Send_Take:SBR22
TITLE=
BEGIN
Network 1
LD     M30.7
A      I3.3
S      M18.7, 1
R      M30.7, 1
Network 2
LD     M30.7
AN     I3.3
AN     I2.2
S      Q1.5, 1
Network 3
LD     M18.7
AN     M3.3
AN     I4.1
S      M21.6, 1
R      M18.7, 1
S      M30.4, 1
R      T118, 1
Network 4
LD     M21.6
AN     I2.2
S      Q1.5, 1
Network 5
LD     Q1.5
A      M21.6
TON    T118, VW36
A      T118
R      T118, 1
S      M29.7, 1
R      M21.6, 1
Network 6
LD     Q1.5
AN     I3.3
AN     M30.3
AN     M30.6
S      M30.6, 1
R      T219, 1
Network 7
LD     M30.6
TON    T219, +2
A      T219
LPS
R      T219, 1
A      I3.3
R      M30.6, 1
LPP
AN     I3.3
S      M30.3, 1
R      M30.6, 1
Network 8
LD     M30.3
A      Q1.5
LD     I3.3
O      I2.2
ALD
R      Q1.5, 1
R      M30.3, 1
R      M21.6, 1
R      M30.6, 1
Network 9
LD     M30.4
AN     I2.2
S      Q1.6, 1
R      T184, 1
R      M30.4, 1
Network 10
LD     Q1.6
AN     M30.5
TON    T184, +20
A      T184
R      T184, 1
S      M30.5, 1
Network 11
LD     M30.5
LD     I4.1
O      M2.3
ALD
R      Q1.6, 1
R      M2.3, 1
R      M30.5, 1
END_SUBROUTINE_BLOCK

DATA_BLOCK_TAB 用户1
BEGIN
VD4000   1.2
VD4004   1.0
VD4008   1.3
VD4012   1.0
VD4016   6.5
VD4020   1.0
VD4024   0.12
VD4028   1.0
VD4032   3.0
VD4036   0.7
VD4044   12.0
VD4048   1.0
VD4052   1.2
VD4070   0.2
VD4074   0.2
VD4078   0.9
VD4086   0.2
VD4090   0.2
VD4094   0.9
VD4102   0.4
VD4106   0.4
VD4110   1.8
VD4118   0.4
VD4122   0.4
VD4126   2.0
VD4196   0.3
VD4200   1.2
VD4204   2.5
VD4212   0.2
VD4216   0.9
VD4220   2.0
VD4228   0.3
VD4232   0.9
VD4236   1.8
VD4244   0.3
VD4248   0.8
VD4252   2.0
VD4260   3.9
VD4264   1.4
VW4500   45
VW4502   40
VW4504   35
VW4506   50
VW4508   35
VW4512   45
VW4514   40
VW4516   35
VW4518   50
VW4520   40
VW4524   99
VW4526   65
VW4528   35
VW4530   60
VW4532   40
VW4536   99
VW4538   65
VW4540   38
VW4542   60
VW4544   28
VW4596   88
VW4598   99
VW4600   55
VW4602   55
VW4604   45
VW4608   90
VW4610   99
VW4612   75
VW4614   45
VW4616   35
VW4620   90
VW4622   95
VW4624   70
VW4626   80
VW4628   45
VW4632   85
VW4634   95
VW4636   80
VW4638   65
VW4640   65
VW4644   65
VW4646   15
VW4650   90
VW4652   99
VW4654   90
VW4656   50
VW4658   25
VW4660   38
VW4662   35
END_DATA_BLOCK_TAB

// (further data pages could not be read)
